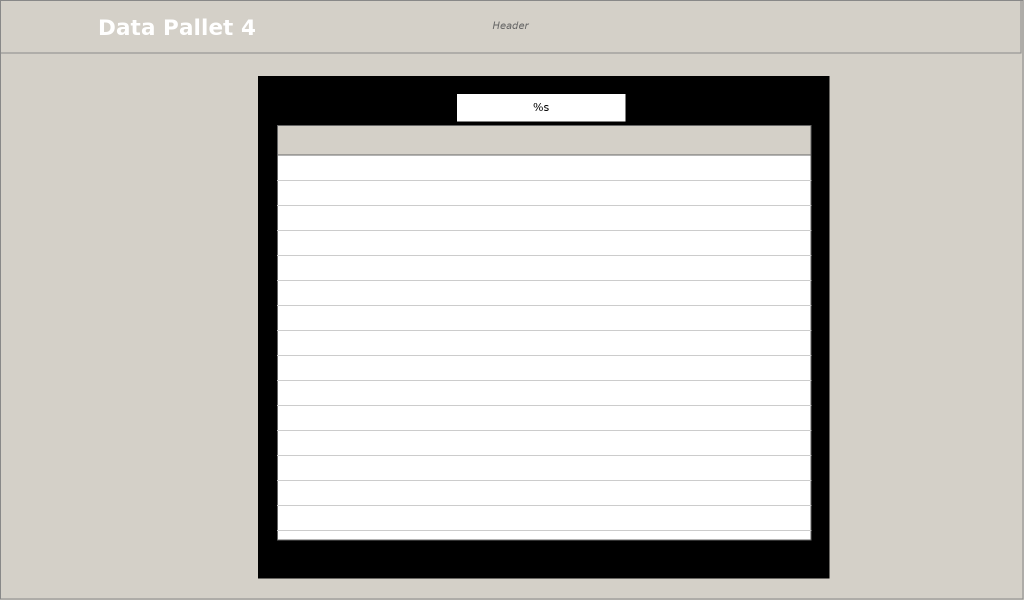
VISUALIZATION DataPallet4  // 1024x600
    Frame (0,-2 1021x55)
        shows Header()
    Label (95,15 250x25), "Data Pallet 4"
    RoundedRectangle (258,76 571x502)
    Table (277,125 534x415), data array: Status_GVL.arDataPallet4
        p3854506369: Status_GVL.arDataPallet4[INDEX].BarcodePallet
        p1892666644: Status_GVL.arDataPallet4[INDEX].BarcodePalletTime
        p338671338: Status_GVL.arPalletizingBuffer[1].EANVariant
        p2170511999: Status_GVL.arPalletizingBuffer[1].CodeVariant
        p3723444502: Status_GVL.arPalletizingBuffer[1].ProductDescription
        p1218418051: Status_GVL.arPalletizingBuffer[1].PalletCreationDate
        p746581629: Status_GVL.arPalletizingBuffer[1].BarcodeProduct
        p3104783080: Status_GVL.arPalletizingBuffer[1].BarcodeProductTime
    RoundedRectangle (456,93 170x29), "%s", text variable: Status_GVL.arPalletID[4]
END_VISUALIZATION

(* stored: Version 1.1.0.1, ProductVersion 3.1.4024.12
   Visu DataPallet4: Id {64802e6d-91fd-4ab6-a8cb-6926b22c5136} *)
